// TIA Portal project "3h sorting" (V16)
// Vorlageprojekt für das Buch mit Zielsystem S7-1200

(* hardware
DEVICE "S7-1200-Station_1"  S7-1200 Station
   slot 0: "Baugruppenträger_0"  Rack  V1.0
   slot 1: "PLC_1"  CPU 1211C DC/DC/DC  6ES7 211-1AE40-0XB0  V4.1
*)

// ===== PLC "PLC_1"  CPU 1211C DC/DC/DC =====

VAR_GLOBAL   // PLC tag table "Standard-Variablentabelle"
   "start" AT %I0.0 : Bool;
   "stop" AT %I0.1 : Bool;
   "sensor 1" AT %I0.2 : Bool;
   "sensor 1(1)" AT %I0.3 : Bool;
   "sensor 2(1)" AT %I0.4 : Bool;
   "sensor 3" AT %I0.5 : Bool;
   "belt convyero (6m) 1" AT %Q0.0 : Bool;
   "belt convyero (4m) 1" AT %Q0.1 : Bool;
   "belt convyero (4m) 2" AT %Q0.2 : Bool;
   "belt convyero (4m) 3" AT %Q0.3 : Bool;
   "pop up wheel sorter 1 (right)" AT %Q0.4 : Bool;
   "pop up wheel sorter 1 (left)" AT %Q0.5 : Bool;
   "pop up wheel sorter 1 (+)" AT %Q0.6 : Bool;
   "loop" AT %M0.0 : Bool;
   "all conveyr" AT %M0.1 : Bool;
   "mm pop up wheel sorter 1 (right)" AT %M0.2 : Bool;
   "mm pop up wheel sorter 1 (+)" AT %M0.3 : Bool;
   "mm pop up wheel sorter 1 (left)" AT %M0.4 : Bool;
END_VAR

FUNCTION "MHJ-PLC-Lab-Function-S71200" : Void   // FC9000, SCL
{ S7_Optimized_Access := 'TRUE' }
VERSION : 0.1
   VAR_TEMP
      rdTimeReturn : Int;
      outputTime : DTL;
      SyncVal : Byte;
      forVal : Int;
      forVal_2 : Int;
      Value : Byte;
   END_VAR
   VAR CONSTANT
      CompVal : Byte := 16#34;
      Value_01 : Byte := 16#11;
      Value_01_DW : DWord := 16#A165_D992;
      Value_02_DW : DWord := 16#58BE_4401;
   END_VAR
BEGIN

   #Value:=PEEK(area := 16#82,
        dbNumber := 0,
        byteOffset := 511);
   #Value := #Value + 1;

   POKE(area := 16#82,
        dbNumber := 0,
        byteOffset := 511,
        value := #Value);

   POKE(area:=16#81,
        dbNumber:=0,
        byteOffset:=1016,
        value:=#Value_01_DW);
   POKE(area := 16#81,
        dbNumber := 0,
        byteOffset := 1020,
        value := #Value_02_DW);

   POKE(area := 16#81,
        dbNumber := 0,
        byteOffset := 511,
        value := B#16#00);

   FOR #forVal := 0 TO 120 DO
       FOR #forVal_2:=0 TO 10 DO
           #rdTimeReturn:=RD_SYS_T(#outputTime);
           #rdTimeReturn := WR_SYS_T(#outputTime);
           #rdTimeReturn := RD_SYS_T(#outputTime);
           #rdTimeReturn := WR_SYS_T(#outputTime);
       END_FOR;
       #SyncVal:= PEEK(area := 16#81,
                      dbNumber := 0,
                      byteOffset := 511);
       IF #SyncVal = #CompVal THEN
          GOTO M_1;
       END_IF;
   END_FOR;
   RETURN;

   M_1:
   POKE(area := 16#81,
        dbNumber := 0,
        byteOffset := 511,
        value := B#16#0);
END_FUNCTION

ORGANIZATION_BLOCK "Main"   // OB1, LAD, ProgramCycle
TITLE = "Main Program Sweep (Cycle)"
{ S7_Optimized_Access := 'TRUE' }
VERSION : 0.1
   VAR_INPUT
      Initial_Call : Bool;   // Initial call of this OB
      Remanence : Bool;   // =True, if remanent data are available
   END_VAR
BEGIN

REGION Network 1: Konnektierungsbaustein für PLC-Lab
   // Im Netzwerk 1 wird der Konnektierungsbaustein für PLC-Lab aufgerufen.
   // Dieser Aufruf darf nicht entfernt werden!
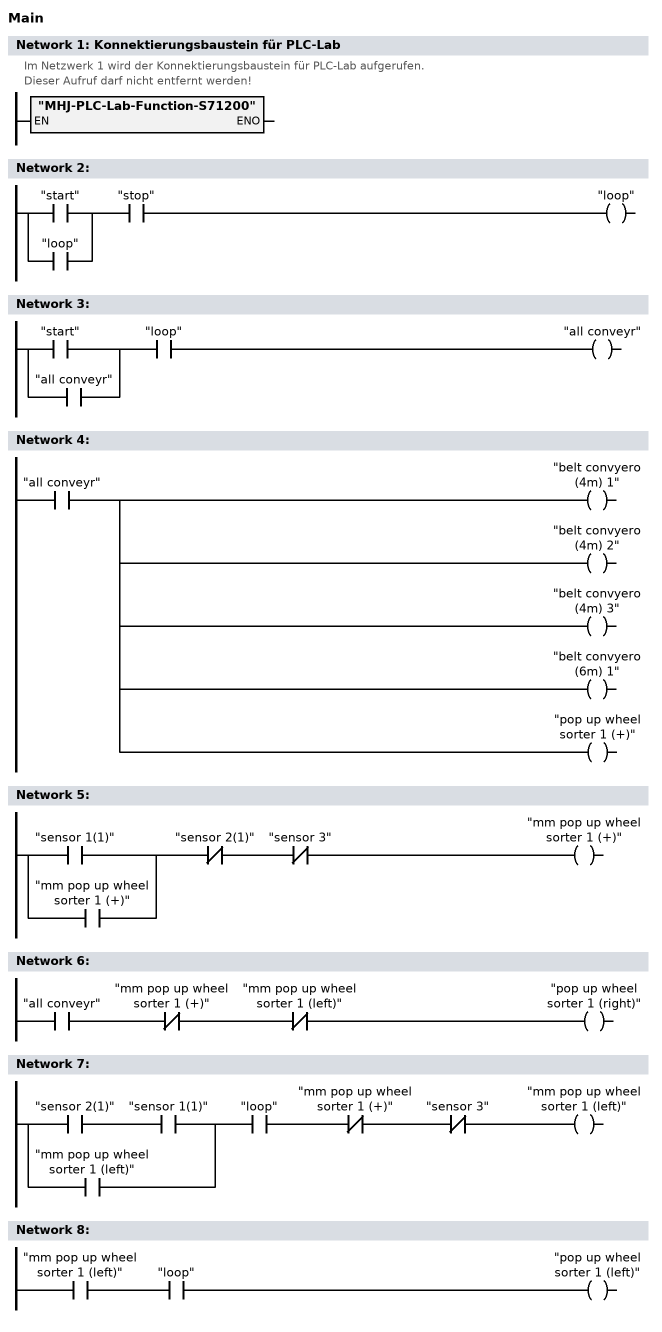
   RUNG wire#powerrail
      "MHJ-PLC-Lab-Function-S71200"()
   END_RUNG
   // the same network as SCL:
   "MHJ-PLC-Lab-Function-S71200"();
END_REGION

REGION Network 2
   RUNG wire#powerrail
      Contact( "start" )
      wire#w1
      Contact( "stop" )
      Coil( "loop" )
   END_RUNG
   RUNG wire#powerrail
      Contact( "loop" )
   END_RUNG wire#w1
   // the same network as SCL:
   "loop" := ("start" OR "loop") AND "stop";
END_REGION

REGION Network 3
   RUNG wire#powerrail
      Contact( "start" )
      wire#w1
      Contact( "loop" )
      Coil( "all conveyr" )
   END_RUNG
   RUNG wire#powerrail
      Contact( "all conveyr" )
   END_RUNG wire#w1
   // the same network as SCL:
   "all conveyr" := ("start" OR "all conveyr") AND "loop";
END_REGION

REGION Network 4
   RUNG wire#powerrail
      Contact( "all conveyr" )
      wire#w1
      Coil( "belt convyero (4m) 1" )
   END_RUNG
   RUNG wire#w1
      Coil( "belt convyero (4m) 2" )
   END_RUNG
   RUNG wire#w1
      Coil( "belt convyero (4m) 3" )
   END_RUNG
   RUNG wire#w1
      Coil( "belt convyero (6m) 1" )
   END_RUNG
   RUNG wire#w1
      Coil( "pop up wheel sorter 1 (+)" )
   END_RUNG
   // the same network as SCL:
   "belt convyero (4m) 1" := "all conveyr";
   "belt convyero (4m) 2" := "all conveyr";
   "belt convyero (4m) 3" := "all conveyr";
   "belt convyero (6m) 1" := "all conveyr";
   "pop up wheel sorter 1 (+)" := "all conveyr";
END_REGION

REGION Network 5
   RUNG wire#powerrail
      Contact( "sensor 1(1)" )
      wire#w1
      I_Contact( "sensor 2(1)" )
      I_Contact( "sensor 3" )
      Coil( "mm pop up wheel sorter 1 (+)" )
   END_RUNG
   RUNG wire#powerrail
      Contact( "mm pop up wheel sorter 1 (+)" )
   END_RUNG wire#w1
   // the same network as SCL:
   "mm pop up wheel sorter 1 (+)" := ("sensor 1(1)" OR "mm pop up wheel sorter 1 (+)") AND NOT "sensor 2(1)" AND NOT "sensor 3";
END_REGION

REGION Network 6
   RUNG wire#powerrail
      Contact( "all conveyr" )
      I_Contact( "mm pop up wheel sorter 1 (+)" )
      I_Contact( "mm pop up wheel sorter 1 (left)" )
      Coil( "pop up wheel sorter 1 (right)" )
   END_RUNG
   // the same network as SCL:
   "pop up wheel sorter 1 (right)" := "all conveyr" AND NOT "mm pop up wheel sorter 1 (+)" AND NOT "mm pop up wheel sorter 1 (left)";
END_REGION

REGION Network 7
   RUNG wire#powerrail
      Contact( "sensor 2(1)" )
      Contact( "sensor 1(1)" )
      wire#w1
      Contact( "loop" )
      I_Contact( "mm pop up wheel sorter 1 (+)" )
      I_Contact( "sensor 3" )
      Coil( "mm pop up wheel sorter 1 (left)" )
   END_RUNG
   RUNG wire#powerrail
      Contact( "mm pop up wheel sorter 1 (left)" )
   END_RUNG wire#w1
   // the same network as SCL:
   "mm pop up wheel sorter 1 (left)" := (("sensor 2(1)" AND "sensor 1(1)") OR "mm pop up wheel sorter 1 (left)") AND "loop" AND NOT "mm pop up wheel sorter 1 (+)" AND NOT "sensor 3";
END_REGION

REGION Network 8
   RUNG wire#powerrail
      Contact( "mm pop up wheel sorter 1 (left)" )
      Contact( "loop" )
      Coil( "pop up wheel sorter 1 (left)" )
   END_RUNG
   // the same network as SCL:
   "pop up wheel sorter 1 (left)" := "mm pop up wheel sorter 1 (left)" AND "loop";
END_REGION
END_ORGANIZATION_BLOCK